% RSLogix 500 project ANALOG1_BAK014.RSS, saved by version 8.40.00.08 %
PROJECT "ANALOG1"    % processor: Bul.1763 MicroLogix 1100 Series B %

PROGRAM FILES
  LAD 2   2 rungs
  LAD 3 "NIVEL"  2 rungs  % Leitura de nivel %
  LAD 4 "BOMBA"  5 rungs  % Comando liga bomba com set e reset %
  LAD 5 "ALARMES"  4 rungs  % Alarmes de nivel alto e baixo %

DATA FILES
  O0 OUTPUT  4 elements
  I1 INPUT  6 elements
  S2 STATUS  66 elements
  B3 BINARY  1 elements
  T4 TIMER  1 elements
  C5 COUNTER  1 elements
  R6 CONTROL  1 elements
  N7 INTEGER  1 elements
  F8 FLOAT  1 elements

LADDER 2
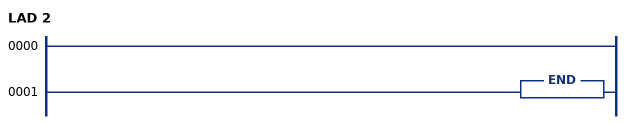
% Rung: 0 %  % edit flag set %
SOR EOR
% Rung: 1 %
SOR END EOR

LADDER 3 "NIVEL"    % Leitura de nivel %
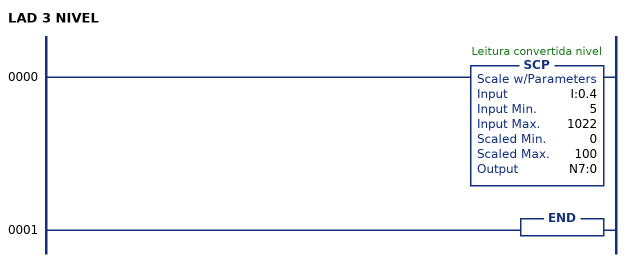
% Rung: 0 %
SOR SCP I:0.4 5 1022 0 100 N7:0 EOR
%   I:0.4  "Entrada analogica nivel" %
%   N7:0  "Leitura convertida nivel" %
% Rung: 1 %
SOR END EOR

LADDER 4 "BOMBA"    % Comando liga bomba com set e reset %
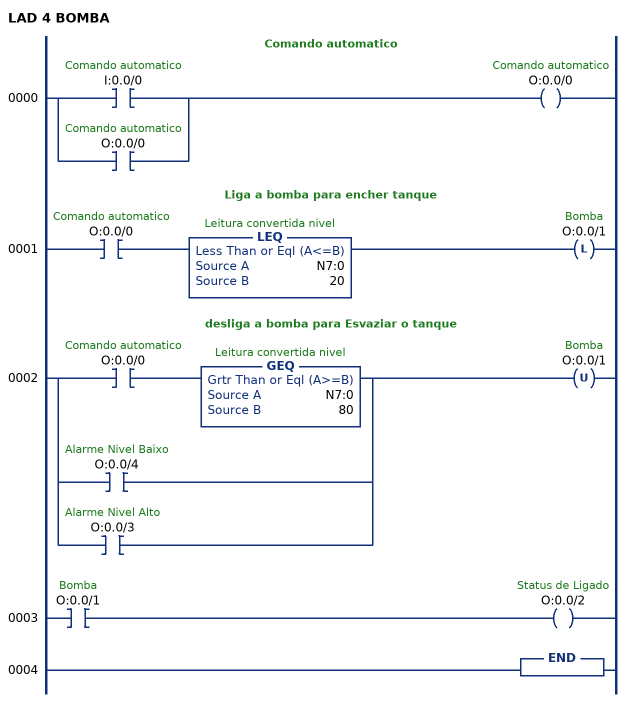
% Rung: 0 %  % edit flag set %
% TITLE: Comando automatico %
SOR BST XIC I:0.0/0 NXB XIC O:0.0/0 BND OTE O:0.0/0 EOR
%   I:0.0/0  "Comando automatico" %
%   O:0.0/0  "Comando automatico" %
% Rung: 1 %  % edit flag set %
% TITLE: Liga a bomba para encher tanque %
SOR XIC O:0.0/0 LEQ N7:0 20 OTL O:0.0/1 EOR
%   O:0.0/0  "Comando automatico" %
%   N7:0  "Leitura convertida nivel" %
%   O:0.0/1  "Bomba" %
% Rung: 2 %  % edit flag set %
% TITLE: desliga a bomba para Esvaziar o tanque %
SOR BST XIC O:0.0/0 GEQ N7:0 80 NXB XIC O:0.0/4 NXB XIC O:0.0/3 BND OTU O:0.0/1 EOR
%   O:0.0/0  "Comando automatico" %
%   N7:0  "Leitura convertida nivel" %
%   O:0.0/4  "Alarme Nivel Baixo" %
%   O:0.0/3  "Alarme Nivel Alto" %
%   O:0.0/1  "Bomba" %
% Rung: 3 %  % edit flag set %
SOR XIC O:0.0/1 OTE O:0.0/2 EOR
%   O:0.0/1  "Bomba" %
%   O:0.0/2  "Status de Ligado" %
% Rung: 4 %
SOR END EOR

LADDER 5 "ALARMES"    % Alarmes de nivel alto e baixo %
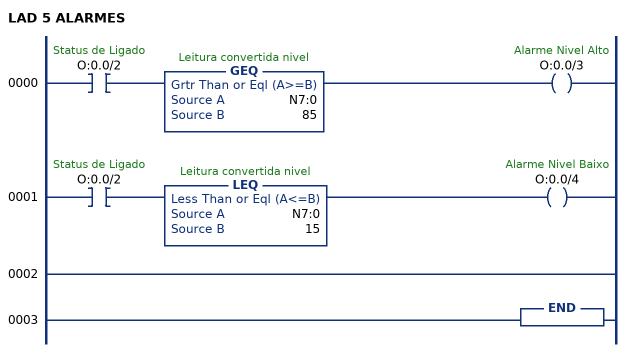
% Rung: 0 %  % edit flag set %
SOR XIC O:0.0/2 GEQ N7:0 85 OTE O:0.0/3 EOR
%   O:0.0/2  "Status de Ligado" %
%   N7:0  "Leitura convertida nivel" %
%   O:0.0/3  "Alarme Nivel Alto" %
% Rung: 1 %  % edit flag set %
SOR XIC O:0.0/2 LEQ N7:0 15 OTE O:0.0/4 EOR
%   O:0.0/2  "Status de Ligado" %
%   N7:0  "Leitura convertida nivel" %
%   O:0.0/4  "Alarme Nivel Baixo" %
% Rung: 2 %  % edit flag set %
SOR EOR
% Rung: 3 %
SOR END EOR

OTHER DOCUMENTED ADDRESSES
  B3:0/0  "desliga bomba"
  F8:0  "Set Point Minimo"
  N7:0/1  "Setpoint Minimo"

COMMENTS NOT ATTACHED TO A CURRENT RUNG
  O:0.0/1: desliga a bomba para Esvaziar o tanque
